% RSLogix 500 project p4.RSS, saved by version 8.10.00.18 %
PROJECT "UNTITLED"    % processor: MicroLogix 1200 %

PROGRAM FILES
  LAD 2   3 rungs
  LAD 3 "IO'S"  7 rungs
  LAD 4 "CONTROL"  6 rungs
  LAD 5 "CYCLE'S"  6 rungs

DATA FILES
  O0 OUTPUT  4 elements
  I1 INPUT  4 elements
  S2 STATUS  66 elements
  B3 BINARY  1 elements
  T4 TIMER  1 elements
  C5 COUNTER  1 elements
  R6 CONTROL  1 elements
  N7 INTEGER  1 elements

LADDER 2
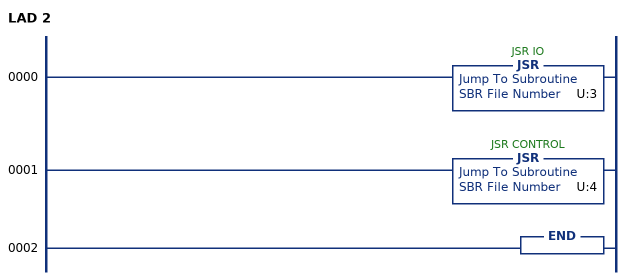
% Rung: 0 %  % edit flag set %
SOR JSR U:3 EOR
%   U:3  "JSR IO" %
% Rung: 1 %  % edit flag set %
SOR JSR U:4 EOR
%   U:4  "JSR CONTROL" %
% Rung: 2 %
SOR END EOR

LADDER 3 "IO'S"
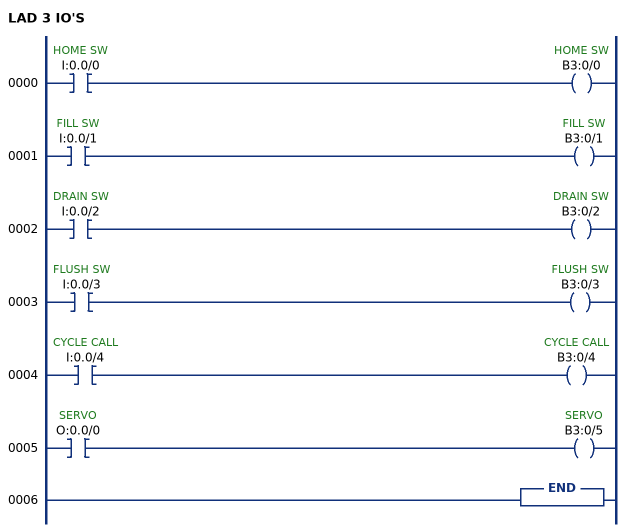
% Rung: 0 %  % edit flag set %
SOR XIC I:0.0/0 OTE B3:0/0 EOR
%   I:0.0/0  "HOME SW" %
%   B3:0/0  "HOME SW" %
% Rung: 1 %  % edit flag set %
SOR XIC I:0.0/1 OTE B3:0/1 EOR
%   I:0.0/1  "FILL SW" %
%   B3:0/1  "FILL SW" %
% Rung: 2 %  % edit flag set %
SOR XIC I:0.0/2 OTE B3:0/2 EOR
%   I:0.0/2  "DRAIN SW" %
%   B3:0/2  "DRAIN SW" %
% Rung: 3 %  % edit flag set %
SOR XIC I:0.0/3 OTE B3:0/3 EOR
%   I:0.0/3  "FLUSH SW" %
%   B3:0/3  "FLUSH SW" %
% Rung: 4 %  % edit flag set %
SOR XIC I:0.0/4 OTE B3:0/4 EOR
%   I:0.0/4  "CYCLE CALL" %
%   B3:0/4  "CYCLE CALL" %
% Rung: 5 %  % edit flag set %
SOR XIC O:0.0/0 OTE B3:0/5 EOR
%   O:0.0/0  "SERVO" %
%   B3:0/5  "SERVO" %
% Rung: 6 %
SOR END EOR

LADDER 4 "CONTROL"
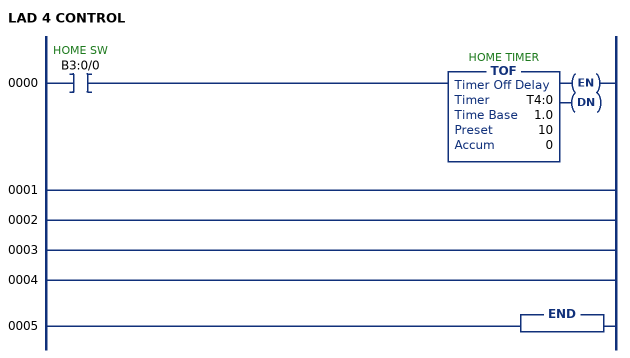
% Rung: 0 %  % edit flag set %
SOR XIC B3:0/0 TOF T4:0 1.0 10 0 EOR
%   B3:0/0  "HOME SW" %
%   T4:0  "HOME TIMER" %
% Rung: 1 %  % edit flag set %
SOR EOR
% Rung: 2 %  % edit flag set %
SOR EOR
% Rung: 3 %  % edit flag set %
SOR EOR
% Rung: 4 %  % edit flag set %
SOR EOR
% Rung: 5 %
SOR END EOR

LADDER 5 "CYCLE'S"
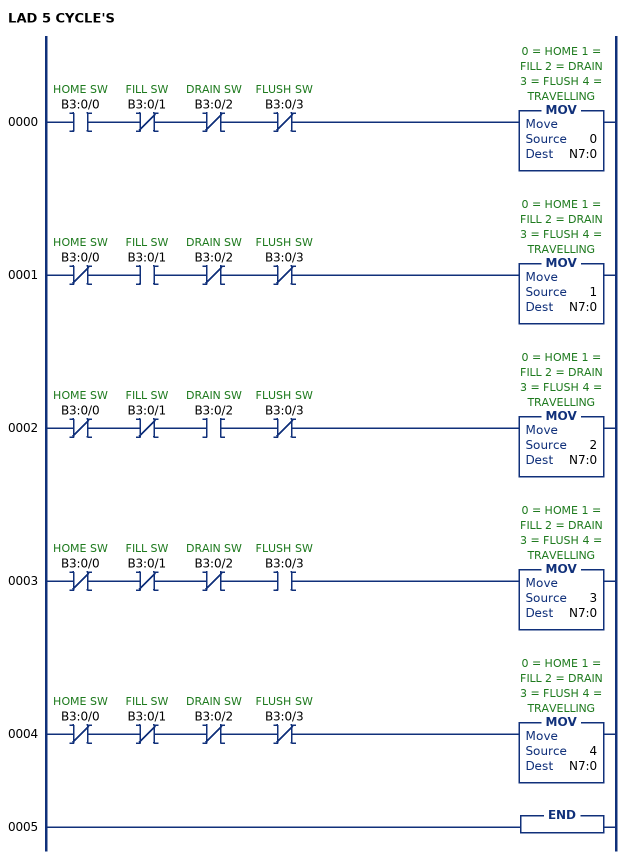
% Rung: 0 %  % edit flag set %
SOR XIC B3:0/0 XIO B3:0/1 XIO B3:0/2 XIO B3:0/3 MOV 0 N7:0 EOR
%   B3:0/0  "HOME SW" %
%   B3:0/1  "FILL SW" %
%   B3:0/2  "DRAIN SW" %
%   B3:0/3  "FLUSH SW" %
%   N7:0  "0 = HOME 1 = FILL 2 = DRAIN 3 = FLUSH 4 = TRAVELLING" %
% Rung: 1 %  % edit flag set %
SOR XIO B3:0/0 XIC B3:0/1 XIO B3:0/2 XIO B3:0/3 MOV 1 N7:0 EOR
%   B3:0/0  "HOME SW" %
%   B3:0/1  "FILL SW" %
%   B3:0/2  "DRAIN SW" %
%   B3:0/3  "FLUSH SW" %
%   N7:0  "0 = HOME 1 = FILL 2 = DRAIN 3 = FLUSH 4 = TRAVELLING" %
% Rung: 2 %  % edit flag set %
SOR XIO B3:0/0 XIO B3:0/1 XIC B3:0/2 XIO B3:0/3 MOV 2 N7:0 EOR
%   B3:0/0  "HOME SW" %
%   B3:0/1  "FILL SW" %
%   B3:0/2  "DRAIN SW" %
%   B3:0/3  "FLUSH SW" %
%   N7:0  "0 = HOME 1 = FILL 2 = DRAIN 3 = FLUSH 4 = TRAVELLING" %
% Rung: 3 %  % edit flag set %
SOR XIO B3:0/0 XIO B3:0/1 XIO B3:0/2 XIC B3:0/3 MOV 3 N7:0 EOR
%   B3:0/0  "HOME SW" %
%   B3:0/1  "FILL SW" %
%   B3:0/2  "DRAIN SW" %
%   B3:0/3  "FLUSH SW" %
%   N7:0  "0 = HOME 1 = FILL 2 = DRAIN 3 = FLUSH 4 = TRAVELLING" %
% Rung: 4 %  % edit flag set %
SOR XIO B3:0/0 XIO B3:0/1 XIO B3:0/2 XIO B3:0/3 MOV 4 N7:0 EOR
%   B3:0/0  "HOME SW" %
%   B3:0/1  "FILL SW" %
%   B3:0/2  "DRAIN SW" %
%   B3:0/3  "FLUSH SW" %
%   N7:0  "0 = HOME 1 = FILL 2 = DRAIN 3 = FLUSH 4 = TRAVELLING" %
% Rung: 5 %
SOR END EOR
